FUNCTION_BLOCK TimeOutBasic (* Basic Function Block Type *)
  (* Standard: 61499-2 *)
  (* Version 0.0, 7/17/2026, Schneider Electric, Template *)
  PACKAGE SE.Nereda;
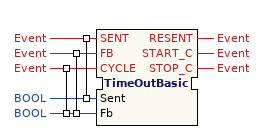
  EVENT_INPUT
    SENT WITH Sent; (* Initialization Request *)
    FB WITH Fb; (* Normal Execution Request *)
    CYCLE WITH Fb;
  END_EVENT
  EVENT_OUTPUT
    RESENT; (* Execution Confirmation *)
    START_C;
    STOP_C;
  END_EVENT
  VAR_INPUT
    Sent : BOOL;
    Fb : BOOL;
  END_VAR
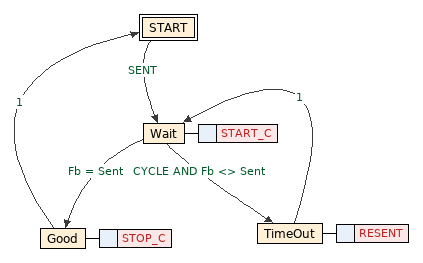
  EC_STATES
    START; (* Initial State *)
    Wait : -> START_C;
    Good : -> STOP_C;
    TimeOut : -> RESENT;
  END_STATES
  EC_TRANSITIONS
    START TO Wait := SENT;
    Wait TO Good := Fb = Sent;
    Wait TO TimeOut := CYCLE AND Fb <> Sent;
    Good TO START := 1;
    TimeOut TO Wait := 1;
  END_TRANSITIONS
END_FUNCTION_BLOCK
